# EPICS substitutions: example-rs232/secage-SE-TDK-RS232App/Db/secage-SE-TDK-RS232.substitutions
file TDK-RS232_Alarm.template
{pattern	{ bl, ta, dn} {SECAGE, SE, TDKR} }

file TDK-RS232_Control.template
{pattern	{ bl, ta, dn} {SECAGE, SE, TDKR} }

file TDK-RS232_General.template
{pattern	{ bl, ta, dn} {SECAGE, SE, TDKR} }
